// TIA Portal V21 export
TYPE "Cambio Altezza"
   STRUCT
      Abilitato : Bool;   // Abilitazione cambio altezza
      "Seq." : Struct
         Step0 : Bool;   // Cambio formato a riposo
         Step1 : Bool;   // Memoria salita per liberare il sensore di massimo formato
         Step2 : Bool;   // Sensore massimo formato liberato
         Step3 : Bool;   // Sensore massimo formato impegnato
         Step4 : Bool;   // Discesa a posizione ricetta
      END_STRUCT;
      x_ENPopUpConferma : Bool;   // Visualizza pop up conferma cambio attrezzatura
      x_PBConferma : Bool;   // PB conferma cambio attrezzatura
   END_STRUCT;
END_TYPE
